(* CoDeSys 2.3 export: ABS_DIFF.EXP *)

(* POU Misc/ABS_DIFF, ST *)
FUNCTION ABS_DIFF : INT
VAR_INPUT
	A: WORD;
	B: WORD;
END_VAR
ABS_DIFF := ABS(WORD_TO_INT(A) - WORD_TO_INT(B));
END_FUNCTION
